// TIA Portal V20 export
// export: Created 2025-12-01T14:57:11.7661616Z, ExportSetting None, DisplayName Totally Integrated Automation Portal, DisplayVersion V20 Update 3, DisplayName TIA Portal Openness, DisplayVersion V20 Update 3, DisplayName TIA Portal Version Control Interface, DisplayVersion V20 Update 3, DisplayName STEP 7 Professional, DisplayVersion V20 Update 3, DisplayName STEP 7 Safety, DisplayVersion V20 Update 2, DisplayName WinCC Basic/Comfort/Advanced, DisplayVersion V20 Update 3, DisplayName WinCC Professional, DisplayVersion V20 Update 3, DisplayName WinCC Unified, DisplayVersion V20 Update 3
FUNCTION "FC920_Registro_Flujos" : Void   // FC920, LAD
TITLE = FC920_Registro_Flujos
{ S7_Optimized_Access := 'FALSE' }
// FC920 Registro Flujos
// stored: AutoNumber false, SetENOAutomatically false
   VAR_INPUT
      Numero_mesa : Int;
   END_VAR
   VAR_TEMP
      cambia_registro : Bool;
      cero : Int;
      retval : Int;
      ROD_CAD : DInt;
      Registro_vacio : Struct
         registro : Array[1..10] of "Registro";
      END_STRUCT;
   END_VAR
   VAR_TEMP   // added for the SCL form of the ladder/FBD networks
      _w1 : Bool;
      _w2 : Bool;
      _w3 : Bool;
      _w4 : Bool;
   END_VAR
BEGIN

REGION Network 1: Inicializacion y cambio de registro registro para poder hacer varios registros
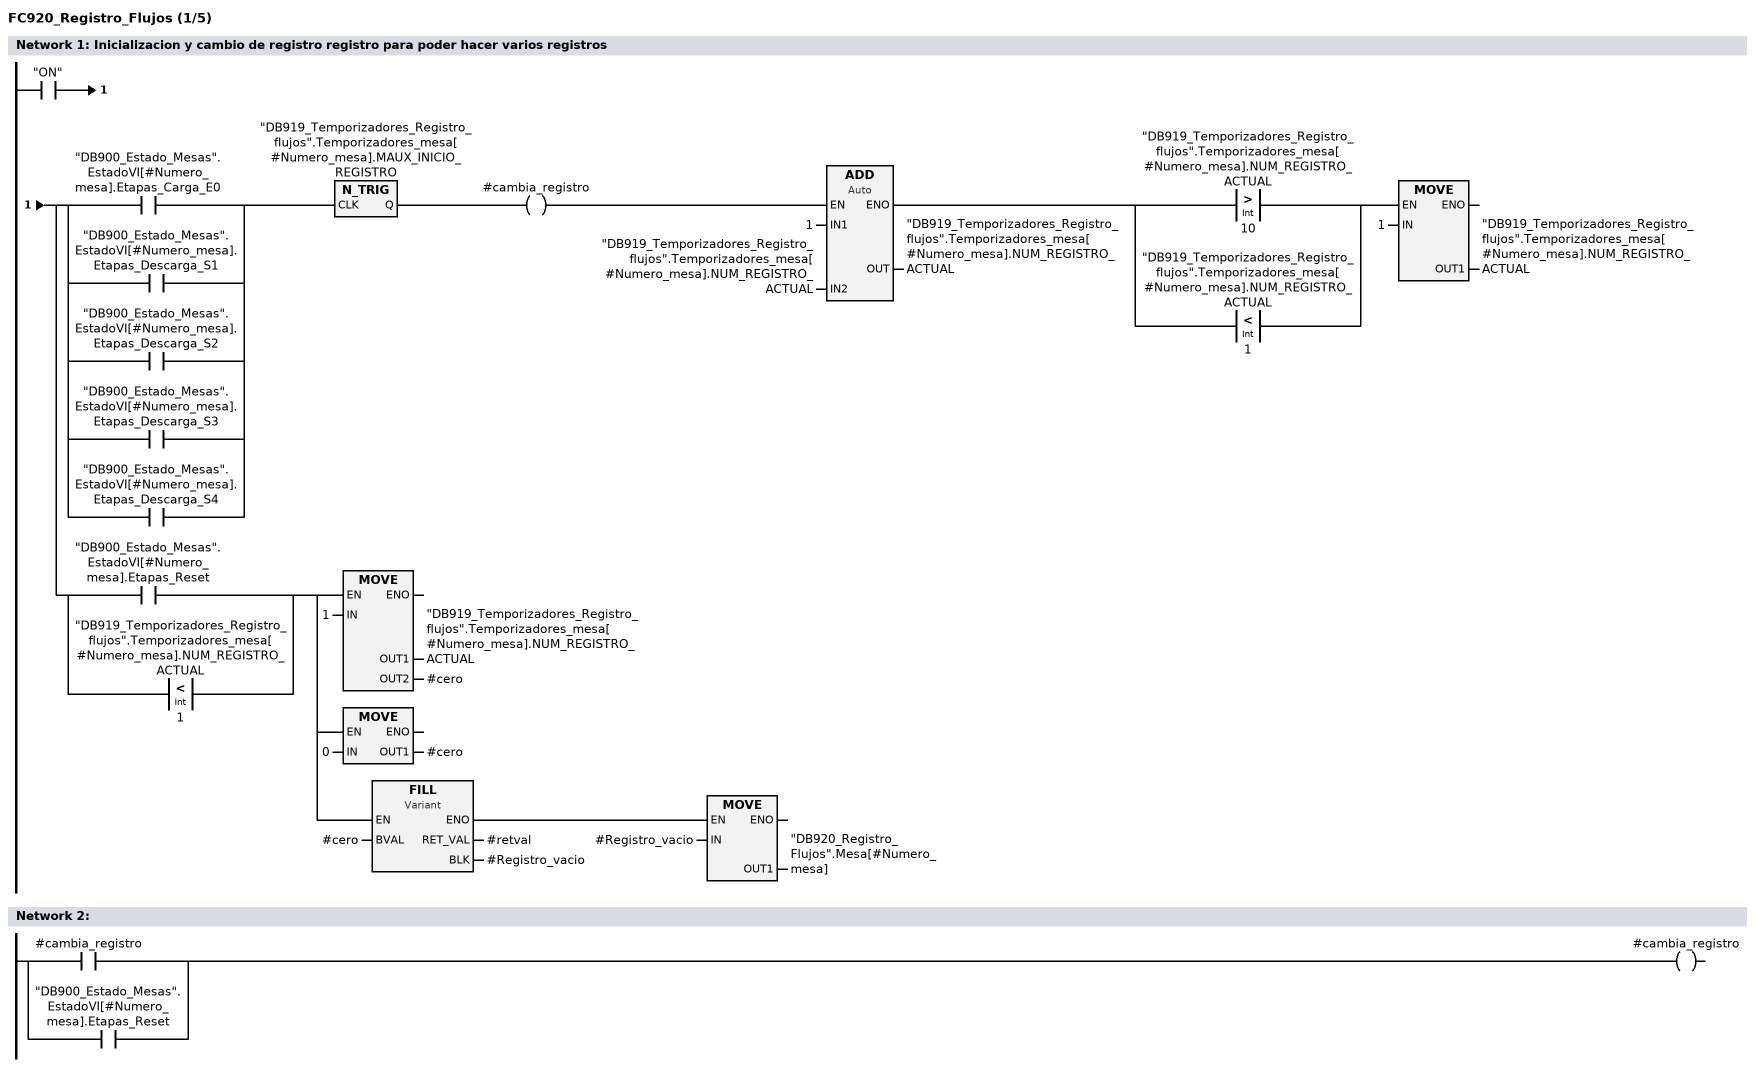
   RUNG wire#powerrail
      Contact( "ON" )
      wire#w1
      Contact( "DB900_Estado_Mesas".EstadoVI[#Numero_mesa].Etapas_Carga_E0 )
      wire#w2
      N_Trig( "DB919_Temporizadores_Registro_flujos".Temporizadores_mesa[#Numero_mesa].MAUX_INICIO_REGISTRO )
      Coil( #cambia_registro )
      Add(in1 := 1, in2 := "DB919_Temporizadores_Registro_flujos".Temporizadores_mesa[#Numero_mesa].NUM_REGISTRO_ACTUAL, out => "DB919_Temporizadores_Registro_flujos".Temporizadores_mesa[#Numero_mesa].NUM_REGISTRO_ACTUAL)
      wire#w3
      { S7_Templates := "SrcType := Int" } GT_Contact(in1 := "DB919_Temporizadores_Registro_flujos".Temporizadores_mesa[#Numero_mesa].NUM_REGISTRO_ACTUAL, in2 := 10)
      wire#w4
      Move(in := 1, out1 => "DB919_Temporizadores_Registro_flujos".Temporizadores_mesa[#Numero_mesa].NUM_REGISTRO_ACTUAL)
   END_RUNG
   RUNG wire#w1
      Contact( "DB900_Estado_Mesas".EstadoVI[#Numero_mesa].Etapas_Descarga_S1 )
   END_RUNG wire#w2
   RUNG wire#w1
      Contact( "DB900_Estado_Mesas".EstadoVI[#Numero_mesa].Etapas_Descarga_S2 )
   END_RUNG wire#w2
   RUNG wire#w1
      Contact( "DB900_Estado_Mesas".EstadoVI[#Numero_mesa].Etapas_Descarga_S3 )
   END_RUNG wire#w2
   RUNG wire#w1
      Contact( "DB900_Estado_Mesas".EstadoVI[#Numero_mesa].Etapas_Descarga_S4 )
   END_RUNG wire#w2
   RUNG wire#w3
      { S7_Templates := "SrcType := Int" } LT_Contact(in1 := "DB919_Temporizadores_Registro_flujos".Temporizadores_mesa[#Numero_mesa].NUM_REGISTRO_ACTUAL, in2 := 1)
   END_RUNG wire#w4
   RUNG wire#w1
      Contact( "DB900_Estado_Mesas".EstadoVI[#Numero_mesa].Etapas_Reset )
      wire#w5
      Move(in := 1, out1 => "DB919_Temporizadores_Registro_flujos".Temporizadores_mesa[#Numero_mesa].NUM_REGISTRO_ACTUAL, out2 => #cero)
   END_RUNG
   RUNG wire#w1
      { S7_Templates := "SrcType := Int" } LT_Contact(in1 := "DB919_Temporizadores_Registro_flujos".Temporizadores_mesa[#Numero_mesa].NUM_REGISTRO_ACTUAL, in2 := 1)
   END_RUNG wire#w5
   RUNG wire#w5
      Move(in := 0, out1 => #cero)
   END_RUNG
   RUNG wire#w5
      { S7_Templates := "ptr_type := Variant" } FILL(BVAL := #cero, RET_VAL => #retval, BLK => #Registro_vacio)
      Move(in := #Registro_vacio, out1 => "DB920_Registro_Flujos".Mesa[#Numero_mesa])
   END_RUNG
   // the same network as SCL:
   #_w1 := "ON" AND ("DB900_Estado_Mesas".EstadoVI[#Numero_mesa].Etapas_Carga_E0 OR "DB900_Estado_Mesas".EstadoVI[#Numero_mesa].Etapas_Descarga_S1 OR "DB900_Estado_Mesas".EstadoVI[#Numero_mesa].Etapas_Descarga_S2 OR "DB900_Estado_Mesas".EstadoVI[#Numero_mesa].Etapas_Descarga_S3 OR "DB900_Estado_Mesas".EstadoVI[#Numero_mesa].Etapas_Descarga_S4);
   #_w2 := NOT #_w1 AND "DB919_Temporizadores_Registro_flujos".Temporizadores_mesa[#Numero_mesa].MAUX_INICIO_REGISTRO;   // falling edge
   "DB919_Temporizadores_Registro_flujos".Temporizadores_mesa[#Numero_mesa].MAUX_INICIO_REGISTRO := #_w1;
   #cambia_registro := #_w2;
   IF #_w2 THEN
       "DB919_Temporizadores_Registro_flujos".Temporizadores_mesa[#Numero_mesa].NUM_REGISTRO_ACTUAL := 1 + "DB919_Temporizadores_Registro_flujos".Temporizadores_mesa[#Numero_mesa].NUM_REGISTRO_ACTUAL;
   END_IF;
   IF #_w2 AND (("DB919_Temporizadores_Registro_flujos".Temporizadores_mesa[#Numero_mesa].NUM_REGISTRO_ACTUAL > 10) OR ("DB919_Temporizadores_Registro_flujos".Temporizadores_mesa[#Numero_mesa].NUM_REGISTRO_ACTUAL < 1)) THEN
       "DB919_Temporizadores_Registro_flujos".Temporizadores_mesa[#Numero_mesa].NUM_REGISTRO_ACTUAL := 1;
   END_IF;
   #_w3 := "ON" AND ("DB900_Estado_Mesas".EstadoVI[#Numero_mesa].Etapas_Reset OR ("DB919_Temporizadores_Registro_flujos".Temporizadores_mesa[#Numero_mesa].NUM_REGISTRO_ACTUAL < 1));
   IF #_w3 THEN
       "DB919_Temporizadores_Registro_flujos".Temporizadores_mesa[#Numero_mesa].NUM_REGISTRO_ACTUAL := 1;
       #cero := 1;
       #cero := 0;
   END_IF;
   #retval := FILL(EN := #_w3, BVAL := #cero, BLK => #Registro_vacio, ENO => #_w4);
   IF #_w4 THEN "DB920_Registro_Flujos".Mesa[#Numero_mesa] := #Registro_vacio; END_IF;
END_REGION

REGION Network 2
   RUNG wire#powerrail
      Contact( #cambia_registro )
      wire#w1
      Coil( #cambia_registro )
   END_RUNG
   RUNG wire#powerrail
      Contact( "DB900_Estado_Mesas".EstadoVI[#Numero_mesa].Etapas_Reset )
   END_RUNG wire#w1
   // the same network as SCL:
   #cambia_registro := #cambia_registro OR "DB900_Estado_Mesas".EstadoVI[#Numero_mesa].Etapas_Reset;
END_REGION

REGION Network 3: Temporizador Etapas de Carga
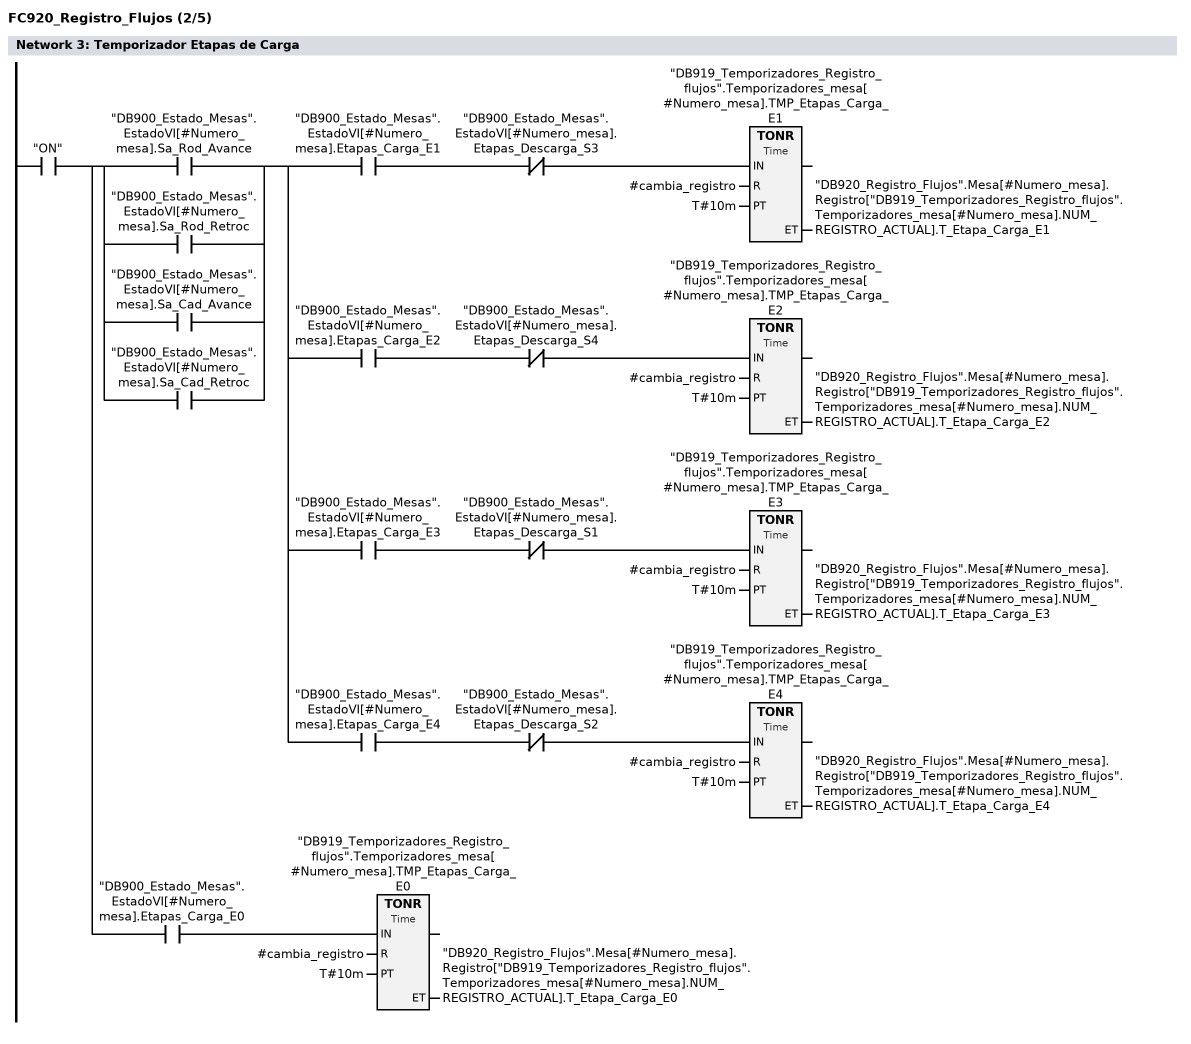
   RUNG wire#powerrail
      Contact( "ON" )
      wire#w1
      Contact( "DB900_Estado_Mesas".EstadoVI[#Numero_mesa].Sa_Rod_Avance )
      wire#w2
      Contact( "DB900_Estado_Mesas".EstadoVI[#Numero_mesa].Etapas_Carga_E1 )
      I_Contact( "DB900_Estado_Mesas".EstadoVI[#Numero_mesa].Etapas_Descarga_S3 )
      { S7_Templates := "time_type := Time" } "DB919_Temporizadores_Registro_flujos".Temporizadores_mesa[#Numero_mesa].TMP_Etapas_Carga_E1.TONR(r := #cambia_registro, pt := T#10m, et => "DB920_Registro_Flujos".Mesa[#Numero_mesa].Registro["DB919_Temporizadores_Registro_flujos".Temporizadores_mesa[#Numero_mesa].NUM_REGISTRO_ACTUAL].T_Etapa_Carga_E1)
   END_RUNG
   RUNG wire#w1
      Contact( "DB900_Estado_Mesas".EstadoVI[#Numero_mesa].Sa_Rod_Retroc )
   END_RUNG wire#w2
   RUNG wire#w1
      Contact( "DB900_Estado_Mesas".EstadoVI[#Numero_mesa].Sa_Cad_Avance )
   END_RUNG wire#w2
   RUNG wire#w1
      Contact( "DB900_Estado_Mesas".EstadoVI[#Numero_mesa].Sa_Cad_Retroc )
   END_RUNG wire#w2
   RUNG wire#w2
      Contact( "DB900_Estado_Mesas".EstadoVI[#Numero_mesa].Etapas_Carga_E2 )
      I_Contact( "DB900_Estado_Mesas".EstadoVI[#Numero_mesa].Etapas_Descarga_S4 )
      { S7_Templates := "time_type := Time" } "DB919_Temporizadores_Registro_flujos".Temporizadores_mesa[#Numero_mesa].TMP_Etapas_Carga_E2.TONR(r := #cambia_registro, pt := T#10m, et => "DB920_Registro_Flujos".Mesa[#Numero_mesa].Registro["DB919_Temporizadores_Registro_flujos".Temporizadores_mesa[#Numero_mesa].NUM_REGISTRO_ACTUAL].T_Etapa_Carga_E2)
   END_RUNG
   RUNG wire#w2
      Contact( "DB900_Estado_Mesas".EstadoVI[#Numero_mesa].Etapas_Carga_E3 )
      I_Contact( "DB900_Estado_Mesas".EstadoVI[#Numero_mesa].Etapas_Descarga_S1 )
      { S7_Templates := "time_type := Time" } "DB919_Temporizadores_Registro_flujos".Temporizadores_mesa[#Numero_mesa].TMP_Etapas_Carga_E3.TONR(r := #cambia_registro, pt := T#10m, et => "DB920_Registro_Flujos".Mesa[#Numero_mesa].Registro["DB919_Temporizadores_Registro_flujos".Temporizadores_mesa[#Numero_mesa].NUM_REGISTRO_ACTUAL].T_Etapa_Carga_E3)
   END_RUNG
   RUNG wire#w2
      Contact( "DB900_Estado_Mesas".EstadoVI[#Numero_mesa].Etapas_Carga_E4 )
      I_Contact( "DB900_Estado_Mesas".EstadoVI[#Numero_mesa].Etapas_Descarga_S2 )
      { S7_Templates := "time_type := Time" } "DB919_Temporizadores_Registro_flujos".Temporizadores_mesa[#Numero_mesa].TMP_Etapas_Carga_E4.TONR(r := #cambia_registro, pt := T#10m, et => "DB920_Registro_Flujos".Mesa[#Numero_mesa].Registro["DB919_Temporizadores_Registro_flujos".Temporizadores_mesa[#Numero_mesa].NUM_REGISTRO_ACTUAL].T_Etapa_Carga_E4)
   END_RUNG
   RUNG wire#w1
      Contact( "DB900_Estado_Mesas".EstadoVI[#Numero_mesa].Etapas_Carga_E0 )
      { S7_Templates := "time_type := Time" } "DB919_Temporizadores_Registro_flujos".Temporizadores_mesa[#Numero_mesa].TMP_Etapas_Carga_E0.TONR(r := #cambia_registro, pt := T#10m, et => "DB920_Registro_Flujos".Mesa[#Numero_mesa].Registro["DB919_Temporizadores_Registro_flujos".Temporizadores_mesa[#Numero_mesa].NUM_REGISTRO_ACTUAL].T_Etapa_Carga_E0)
   END_RUNG
   // the same network as SCL:
   #_w1 := "ON" AND ("DB900_Estado_Mesas".EstadoVI[#Numero_mesa].Sa_Rod_Avance OR "DB900_Estado_Mesas".EstadoVI[#Numero_mesa].Sa_Rod_Retroc OR "DB900_Estado_Mesas".EstadoVI[#Numero_mesa].Sa_Cad_Avance OR "DB900_Estado_Mesas".EstadoVI[#Numero_mesa].Sa_Cad_Retroc);
   "DB919_Temporizadores_Registro_flujos".Temporizadores_mesa[#Numero_mesa].TMP_Etapas_Carga_E1.TONR(IN := #_w1 AND "DB900_Estado_Mesas".EstadoVI[#Numero_mesa].Etapas_Carga_E1 AND NOT "DB900_Estado_Mesas".EstadoVI[#Numero_mesa].Etapas_Descarga_S3,
                           R := #cambia_registro,
                           PT := T#10m,
                           ET => "DB920_Registro_Flujos".Mesa[#Numero_mesa].Registro["DB919_Temporizadores_Registro_flujos".Temporizadores_mesa[#Numero_mesa].NUM_REGISTRO_ACTUAL].T_Etapa_Carga_E1);
   "DB919_Temporizadores_Registro_flujos".Temporizadores_mesa[#Numero_mesa].TMP_Etapas_Carga_E2.TONR(IN := #_w1 AND "DB900_Estado_Mesas".EstadoVI[#Numero_mesa].Etapas_Carga_E2 AND NOT "DB900_Estado_Mesas".EstadoVI[#Numero_mesa].Etapas_Descarga_S4,
                           R := #cambia_registro,
                           PT := T#10m,
                           ET => "DB920_Registro_Flujos".Mesa[#Numero_mesa].Registro["DB919_Temporizadores_Registro_flujos".Temporizadores_mesa[#Numero_mesa].NUM_REGISTRO_ACTUAL].T_Etapa_Carga_E2);
   "DB919_Temporizadores_Registro_flujos".Temporizadores_mesa[#Numero_mesa].TMP_Etapas_Carga_E3.TONR(IN := #_w1 AND "DB900_Estado_Mesas".EstadoVI[#Numero_mesa].Etapas_Carga_E3 AND NOT "DB900_Estado_Mesas".EstadoVI[#Numero_mesa].Etapas_Descarga_S1,
                           R := #cambia_registro,
                           PT := T#10m,
                           ET => "DB920_Registro_Flujos".Mesa[#Numero_mesa].Registro["DB919_Temporizadores_Registro_flujos".Temporizadores_mesa[#Numero_mesa].NUM_REGISTRO_ACTUAL].T_Etapa_Carga_E3);
   "DB919_Temporizadores_Registro_flujos".Temporizadores_mesa[#Numero_mesa].TMP_Etapas_Carga_E4.TONR(IN := #_w1 AND "DB900_Estado_Mesas".EstadoVI[#Numero_mesa].Etapas_Carga_E4 AND NOT "DB900_Estado_Mesas".EstadoVI[#Numero_mesa].Etapas_Descarga_S2,
                           R := #cambia_registro,
                           PT := T#10m,
                           ET => "DB920_Registro_Flujos".Mesa[#Numero_mesa].Registro["DB919_Temporizadores_Registro_flujos".Temporizadores_mesa[#Numero_mesa].NUM_REGISTRO_ACTUAL].T_Etapa_Carga_E4);
   "DB919_Temporizadores_Registro_flujos".Temporizadores_mesa[#Numero_mesa].TMP_Etapas_Carga_E0.TONR(IN := "ON" AND "DB900_Estado_Mesas".EstadoVI[#Numero_mesa].Etapas_Carga_E0,
                           R := #cambia_registro,
                           PT := T#10m,
                           ET => "DB920_Registro_Flujos".Mesa[#Numero_mesa].Registro["DB919_Temporizadores_Registro_flujos".Temporizadores_mesa[#Numero_mesa].NUM_REGISTRO_ACTUAL].T_Etapa_Carga_E0);
END_REGION

REGION Network 4: Temporizador Etapas de Descarga
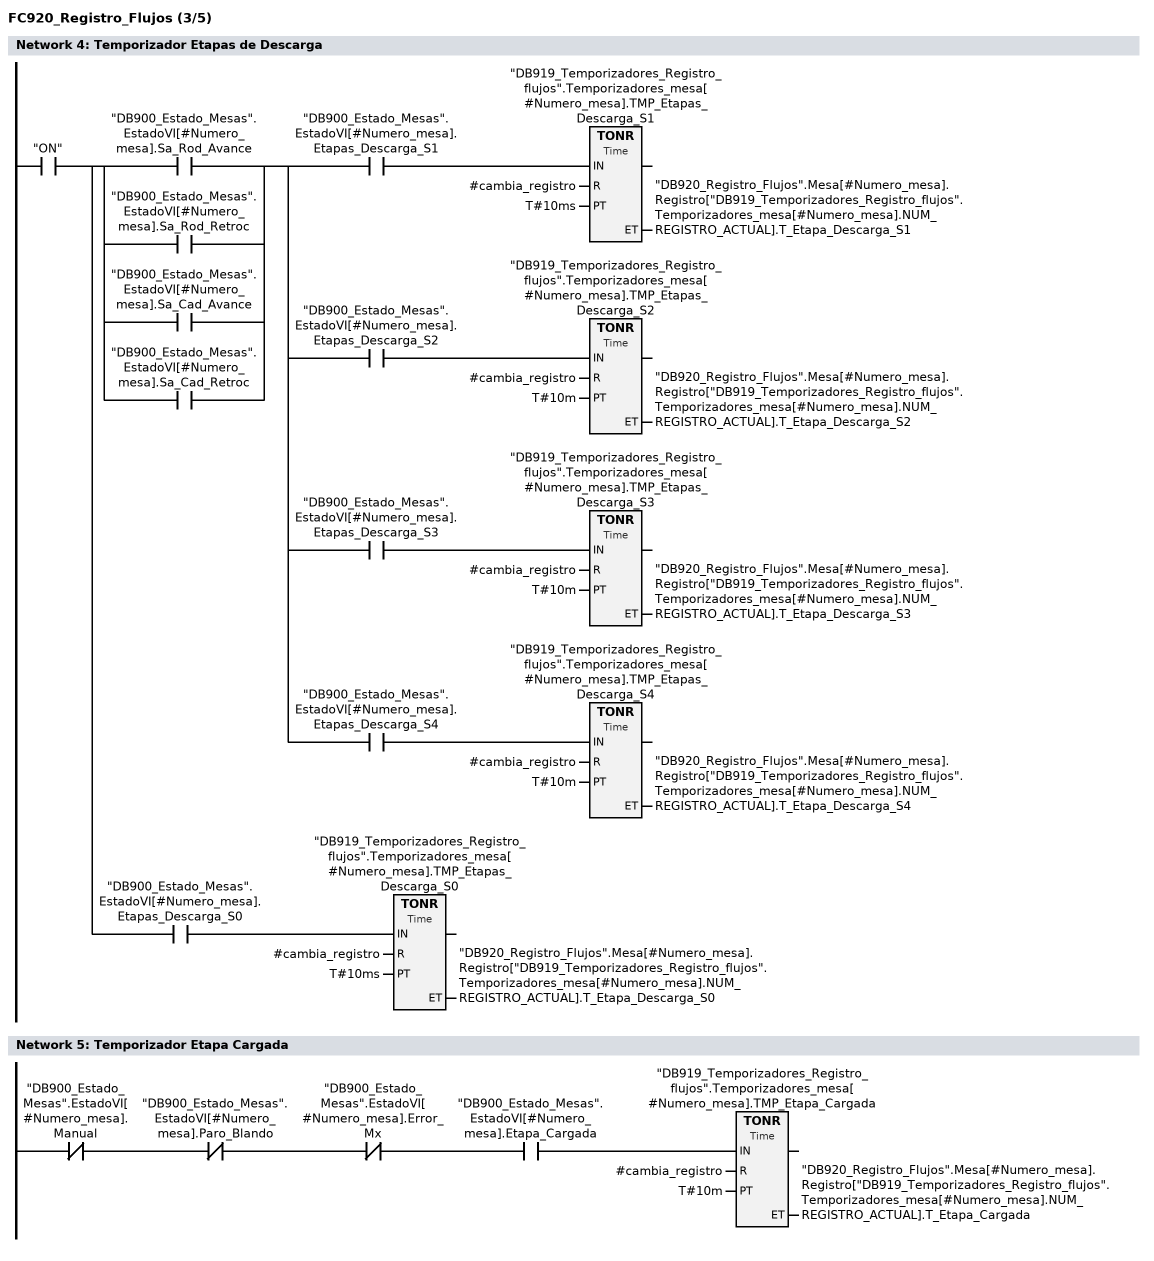
   RUNG wire#powerrail
      Contact( "ON" )
      wire#w1
      Contact( "DB900_Estado_Mesas".EstadoVI[#Numero_mesa].Sa_Rod_Avance )
      wire#w2
      Contact( "DB900_Estado_Mesas".EstadoVI[#Numero_mesa].Etapas_Descarga_S1 )
      { S7_Templates := "time_type := Time" } "DB919_Temporizadores_Registro_flujos".Temporizadores_mesa[#Numero_mesa].TMP_Etapas_Descarga_S1.TONR(r := #cambia_registro, pt := T#10ms, et => "DB920_Registro_Flujos".Mesa[#Numero_mesa].Registro["DB919_Temporizadores_Registro_flujos".Temporizadores_mesa[#Numero_mesa].NUM_REGISTRO_ACTUAL].T_Etapa_Descarga_S1)
   END_RUNG
   RUNG wire#w1
      Contact( "DB900_Estado_Mesas".EstadoVI[#Numero_mesa].Sa_Rod_Retroc )
   END_RUNG wire#w2
   RUNG wire#w1
      Contact( "DB900_Estado_Mesas".EstadoVI[#Numero_mesa].Sa_Cad_Avance )
   END_RUNG wire#w2
   RUNG wire#w1
      Contact( "DB900_Estado_Mesas".EstadoVI[#Numero_mesa].Sa_Cad_Retroc )
   END_RUNG wire#w2
   RUNG wire#w2
      Contact( "DB900_Estado_Mesas".EstadoVI[#Numero_mesa].Etapas_Descarga_S2 )
      { S7_Templates := "time_type := Time" } "DB919_Temporizadores_Registro_flujos".Temporizadores_mesa[#Numero_mesa].TMP_Etapas_Descarga_S2.TONR(r := #cambia_registro, pt := T#10m, et => "DB920_Registro_Flujos".Mesa[#Numero_mesa].Registro["DB919_Temporizadores_Registro_flujos".Temporizadores_mesa[#Numero_mesa].NUM_REGISTRO_ACTUAL].T_Etapa_Descarga_S2)
   END_RUNG
   RUNG wire#w2
      Contact( "DB900_Estado_Mesas".EstadoVI[#Numero_mesa].Etapas_Descarga_S3 )
      { S7_Templates := "time_type := Time" } "DB919_Temporizadores_Registro_flujos".Temporizadores_mesa[#Numero_mesa].TMP_Etapas_Descarga_S3.TONR(r := #cambia_registro, pt := T#10m, et => "DB920_Registro_Flujos".Mesa[#Numero_mesa].Registro["DB919_Temporizadores_Registro_flujos".Temporizadores_mesa[#Numero_mesa].NUM_REGISTRO_ACTUAL].T_Etapa_Descarga_S3)
   END_RUNG
   RUNG wire#w2
      Contact( "DB900_Estado_Mesas".EstadoVI[#Numero_mesa].Etapas_Descarga_S4 )
      { S7_Templates := "time_type := Time" } "DB919_Temporizadores_Registro_flujos".Temporizadores_mesa[#Numero_mesa].TMP_Etapas_Descarga_S4.TONR(r := #cambia_registro, pt := T#10m, et => "DB920_Registro_Flujos".Mesa[#Numero_mesa].Registro["DB919_Temporizadores_Registro_flujos".Temporizadores_mesa[#Numero_mesa].NUM_REGISTRO_ACTUAL].T_Etapa_Descarga_S4)
   END_RUNG
   RUNG wire#w1
      Contact( "DB900_Estado_Mesas".EstadoVI[#Numero_mesa].Etapas_Descarga_S0 )
      { S7_Templates := "time_type := Time" } "DB919_Temporizadores_Registro_flujos".Temporizadores_mesa[#Numero_mesa].TMP_Etapas_Descarga_S0.TONR(r := #cambia_registro, pt := T#10ms, et => "DB920_Registro_Flujos".Mesa[#Numero_mesa].Registro["DB919_Temporizadores_Registro_flujos".Temporizadores_mesa[#Numero_mesa].NUM_REGISTRO_ACTUAL].T_Etapa_Descarga_S0)
   END_RUNG
   // the same network as SCL:
   #_w1 := "ON" AND ("DB900_Estado_Mesas".EstadoVI[#Numero_mesa].Sa_Rod_Avance OR "DB900_Estado_Mesas".EstadoVI[#Numero_mesa].Sa_Rod_Retroc OR "DB900_Estado_Mesas".EstadoVI[#Numero_mesa].Sa_Cad_Avance OR "DB900_Estado_Mesas".EstadoVI[#Numero_mesa].Sa_Cad_Retroc);
   "DB919_Temporizadores_Registro_flujos".Temporizadores_mesa[#Numero_mesa].TMP_Etapas_Descarga_S1.TONR(IN := #_w1 AND "DB900_Estado_Mesas".EstadoVI[#Numero_mesa].Etapas_Descarga_S1,
                           R := #cambia_registro,
                           PT := T#10ms,
                           ET => "DB920_Registro_Flujos".Mesa[#Numero_mesa].Registro["DB919_Temporizadores_Registro_flujos".Temporizadores_mesa[#Numero_mesa].NUM_REGISTRO_ACTUAL].T_Etapa_Descarga_S1);
   "DB919_Temporizadores_Registro_flujos".Temporizadores_mesa[#Numero_mesa].TMP_Etapas_Descarga_S2.TONR(IN := #_w1 AND "DB900_Estado_Mesas".EstadoVI[#Numero_mesa].Etapas_Descarga_S2,
                           R := #cambia_registro,
                           PT := T#10m,
                           ET => "DB920_Registro_Flujos".Mesa[#Numero_mesa].Registro["DB919_Temporizadores_Registro_flujos".Temporizadores_mesa[#Numero_mesa].NUM_REGISTRO_ACTUAL].T_Etapa_Descarga_S2);
   "DB919_Temporizadores_Registro_flujos".Temporizadores_mesa[#Numero_mesa].TMP_Etapas_Descarga_S3.TONR(IN := #_w1 AND "DB900_Estado_Mesas".EstadoVI[#Numero_mesa].Etapas_Descarga_S3,
                           R := #cambia_registro,
                           PT := T#10m,
                           ET => "DB920_Registro_Flujos".Mesa[#Numero_mesa].Registro["DB919_Temporizadores_Registro_flujos".Temporizadores_mesa[#Numero_mesa].NUM_REGISTRO_ACTUAL].T_Etapa_Descarga_S3);
   "DB919_Temporizadores_Registro_flujos".Temporizadores_mesa[#Numero_mesa].TMP_Etapas_Descarga_S4.TONR(IN := #_w1 AND "DB900_Estado_Mesas".EstadoVI[#Numero_mesa].Etapas_Descarga_S4,
                           R := #cambia_registro,
                           PT := T#10m,
                           ET => "DB920_Registro_Flujos".Mesa[#Numero_mesa].Registro["DB919_Temporizadores_Registro_flujos".Temporizadores_mesa[#Numero_mesa].NUM_REGISTRO_ACTUAL].T_Etapa_Descarga_S4);
   "DB919_Temporizadores_Registro_flujos".Temporizadores_mesa[#Numero_mesa].TMP_Etapas_Descarga_S0.TONR(IN := "ON" AND "DB900_Estado_Mesas".EstadoVI[#Numero_mesa].Etapas_Descarga_S0,
                           R := #cambia_registro,
                           PT := T#10ms,
                           ET => "DB920_Registro_Flujos".Mesa[#Numero_mesa].Registro["DB919_Temporizadores_Registro_flujos".Temporizadores_mesa[#Numero_mesa].NUM_REGISTRO_ACTUAL].T_Etapa_Descarga_S0);
END_REGION

REGION Network 5: Temporizador Etapa Cargada
   RUNG wire#powerrail
      I_Contact( "DB900_Estado_Mesas".EstadoVI[#Numero_mesa].Manual )
      I_Contact( "DB900_Estado_Mesas".EstadoVI[#Numero_mesa].Paro_Blando )
      I_Contact( "DB900_Estado_Mesas".EstadoVI[#Numero_mesa].Error_Mx )
      Contact( "DB900_Estado_Mesas".EstadoVI[#Numero_mesa].Etapa_Cargada )
      { S7_Templates := "time_type := Time" } "DB919_Temporizadores_Registro_flujos".Temporizadores_mesa[#Numero_mesa].TMP_Etapa_Cargada.TONR(r := #cambia_registro, pt := T#10m, et => "DB920_Registro_Flujos".Mesa[#Numero_mesa].Registro["DB919_Temporizadores_Registro_flujos".Temporizadores_mesa[#Numero_mesa].NUM_REGISTRO_ACTUAL].T_Etapa_Cargada)
   END_RUNG
   // the same network as SCL:
   "DB919_Temporizadores_Registro_flujos".Temporizadores_mesa[#Numero_mesa].TMP_Etapa_Cargada.TONR(IN := NOT "DB900_Estado_Mesas".EstadoVI[#Numero_mesa].Manual AND NOT "DB900_Estado_Mesas".EstadoVI[#Numero_mesa].Paro_Blando AND NOT "DB900_Estado_Mesas".EstadoVI[#Numero_mesa].Error_Mx AND "DB900_Estado_Mesas".EstadoVI[#Numero_mesa].Etapa_Cargada,
                           R := #cambia_registro,
                           PT := T#10m,
                           ET => "DB920_Registro_Flujos".Mesa[#Numero_mesa].Registro["DB919_Temporizadores_Registro_flujos".Temporizadores_mesa[#Numero_mesa].NUM_REGISTRO_ACTUAL].T_Etapa_Cargada);
END_REGION

REGION Network 6: Temporizador Avance/Retroceso Rodillos
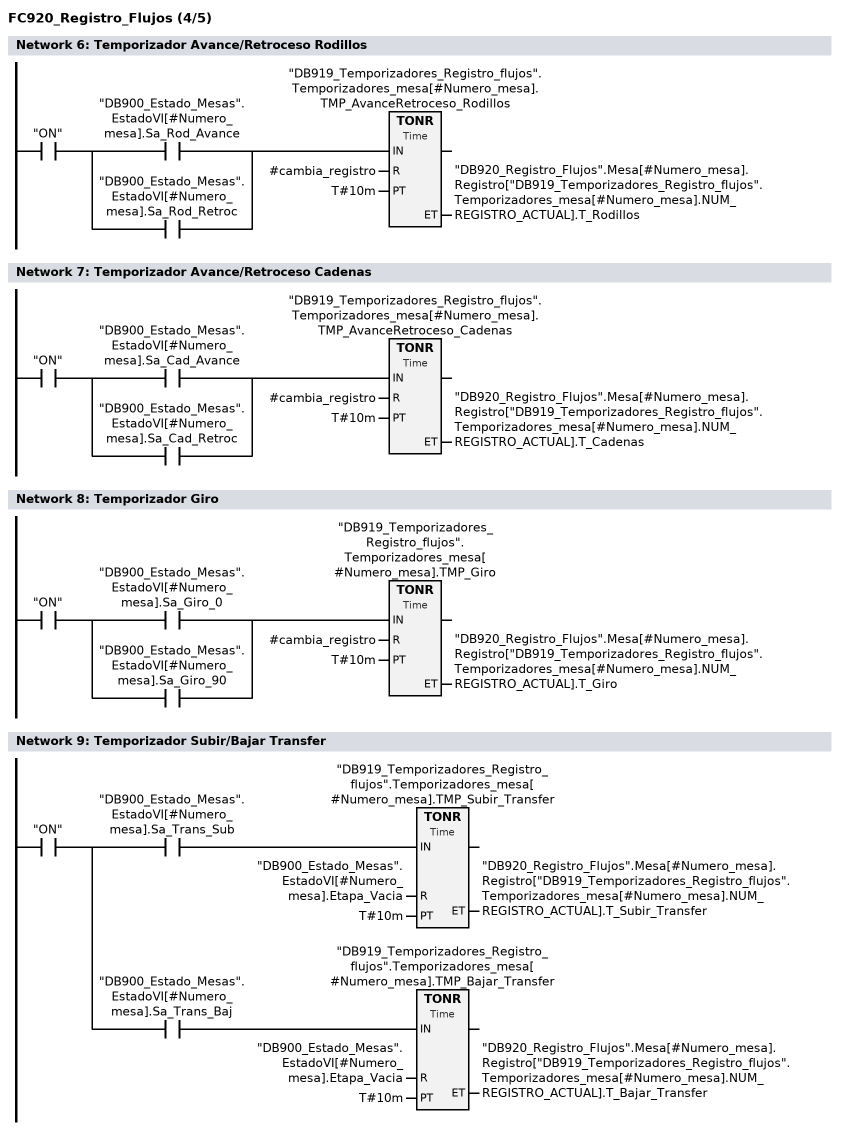
   RUNG wire#powerrail
      Contact( "ON" )
      wire#w1
      Contact( "DB900_Estado_Mesas".EstadoVI[#Numero_mesa].Sa_Rod_Avance )
      wire#w2
      { S7_Templates := "time_type := Time" } "DB919_Temporizadores_Registro_flujos".Temporizadores_mesa[#Numero_mesa].TMP_AvanceRetroceso_Rodillos.TONR(r := #cambia_registro, pt := T#10m, et => "DB920_Registro_Flujos".Mesa[#Numero_mesa].Registro["DB919_Temporizadores_Registro_flujos".Temporizadores_mesa[#Numero_mesa].NUM_REGISTRO_ACTUAL].T_Rodillos)
   END_RUNG
   RUNG wire#w1
      Contact( "DB900_Estado_Mesas".EstadoVI[#Numero_mesa].Sa_Rod_Retroc )
   END_RUNG wire#w2
   // the same network as SCL:
   "DB919_Temporizadores_Registro_flujos".Temporizadores_mesa[#Numero_mesa].TMP_AvanceRetroceso_Rodillos.TONR(IN := "ON" AND ("DB900_Estado_Mesas".EstadoVI[#Numero_mesa].Sa_Rod_Avance OR "DB900_Estado_Mesas".EstadoVI[#Numero_mesa].Sa_Rod_Retroc),
                           R := #cambia_registro,
                           PT := T#10m,
                           ET => "DB920_Registro_Flujos".Mesa[#Numero_mesa].Registro["DB919_Temporizadores_Registro_flujos".Temporizadores_mesa[#Numero_mesa].NUM_REGISTRO_ACTUAL].T_Rodillos);
END_REGION

REGION Network 7: Temporizador Avance/Retroceso Cadenas
   RUNG wire#powerrail
      Contact( "ON" )
      wire#w1
      Contact( "DB900_Estado_Mesas".EstadoVI[#Numero_mesa].Sa_Cad_Avance )
      wire#w2
      { S7_Templates := "time_type := Time" } "DB919_Temporizadores_Registro_flujos".Temporizadores_mesa[#Numero_mesa].TMP_AvanceRetroceso_Cadenas.TONR(r := #cambia_registro, pt := T#10m, et => "DB920_Registro_Flujos".Mesa[#Numero_mesa].Registro["DB919_Temporizadores_Registro_flujos".Temporizadores_mesa[#Numero_mesa].NUM_REGISTRO_ACTUAL].T_Cadenas)
   END_RUNG
   RUNG wire#w1
      Contact( "DB900_Estado_Mesas".EstadoVI[#Numero_mesa].Sa_Cad_Retroc )
   END_RUNG wire#w2
   // the same network as SCL:
   "DB919_Temporizadores_Registro_flujos".Temporizadores_mesa[#Numero_mesa].TMP_AvanceRetroceso_Cadenas.TONR(IN := "ON" AND ("DB900_Estado_Mesas".EstadoVI[#Numero_mesa].Sa_Cad_Avance OR "DB900_Estado_Mesas".EstadoVI[#Numero_mesa].Sa_Cad_Retroc),
                           R := #cambia_registro,
                           PT := T#10m,
                           ET => "DB920_Registro_Flujos".Mesa[#Numero_mesa].Registro["DB919_Temporizadores_Registro_flujos".Temporizadores_mesa[#Numero_mesa].NUM_REGISTRO_ACTUAL].T_Cadenas);
END_REGION

REGION Network 8: Temporizador Giro
   RUNG wire#powerrail
      Contact( "ON" )
      wire#w1
      Contact( "DB900_Estado_Mesas".EstadoVI[#Numero_mesa].Sa_Giro_0 )
      wire#w2
      { S7_Templates := "time_type := Time" } "DB919_Temporizadores_Registro_flujos".Temporizadores_mesa[#Numero_mesa].TMP_Giro.TONR(r := #cambia_registro, pt := T#10m, et => "DB920_Registro_Flujos".Mesa[#Numero_mesa].Registro["DB919_Temporizadores_Registro_flujos".Temporizadores_mesa[#Numero_mesa].NUM_REGISTRO_ACTUAL].T_Giro)
   END_RUNG
   RUNG wire#w1
      Contact( "DB900_Estado_Mesas".EstadoVI[#Numero_mesa].Sa_Giro_90 )
   END_RUNG wire#w2
   // the same network as SCL:
   "DB919_Temporizadores_Registro_flujos".Temporizadores_mesa[#Numero_mesa].TMP_Giro.TONR(IN := "ON" AND ("DB900_Estado_Mesas".EstadoVI[#Numero_mesa].Sa_Giro_0 OR "DB900_Estado_Mesas".EstadoVI[#Numero_mesa].Sa_Giro_90),
                           R := #cambia_registro,
                           PT := T#10m,
                           ET => "DB920_Registro_Flujos".Mesa[#Numero_mesa].Registro["DB919_Temporizadores_Registro_flujos".Temporizadores_mesa[#Numero_mesa].NUM_REGISTRO_ACTUAL].T_Giro);
END_REGION

REGION Network 9: Temporizador Subir/Bajar Transfer
   RUNG wire#powerrail
      Contact( "ON" )
      wire#w1
      Contact( "DB900_Estado_Mesas".EstadoVI[#Numero_mesa].Sa_Trans_Sub )
      { S7_Templates := "time_type := Time" } "DB919_Temporizadores_Registro_flujos".Temporizadores_mesa[#Numero_mesa].TMP_Subir_Transfer.TONR(r := "DB900_Estado_Mesas".EstadoVI[#Numero_mesa].Etapa_Vacia, pt := T#10m, et => "DB920_Registro_Flujos".Mesa[#Numero_mesa].Registro["DB919_Temporizadores_Registro_flujos".Temporizadores_mesa[#Numero_mesa].NUM_REGISTRO_ACTUAL].T_Subir_Transfer)
   END_RUNG
   RUNG wire#w1
      Contact( "DB900_Estado_Mesas".EstadoVI[#Numero_mesa].Sa_Trans_Baj )
      { S7_Templates := "time_type := Time" } "DB919_Temporizadores_Registro_flujos".Temporizadores_mesa[#Numero_mesa].TMP_Bajar_Transfer.TONR(r := "DB900_Estado_Mesas".EstadoVI[#Numero_mesa].Etapa_Vacia, pt := T#10m, et => "DB920_Registro_Flujos".Mesa[#Numero_mesa].Registro["DB919_Temporizadores_Registro_flujos".Temporizadores_mesa[#Numero_mesa].NUM_REGISTRO_ACTUAL].T_Bajar_Transfer)
   END_RUNG
   // the same network as SCL:
   "DB919_Temporizadores_Registro_flujos".Temporizadores_mesa[#Numero_mesa].TMP_Subir_Transfer.TONR(IN := "ON" AND "DB900_Estado_Mesas".EstadoVI[#Numero_mesa].Sa_Trans_Sub,
                           R := "DB900_Estado_Mesas".EstadoVI[#Numero_mesa].Etapa_Vacia,
                           PT := T#10m,
                           ET => "DB920_Registro_Flujos".Mesa[#Numero_mesa].Registro["DB919_Temporizadores_Registro_flujos".Temporizadores_mesa[#Numero_mesa].NUM_REGISTRO_ACTUAL].T_Subir_Transfer);
   "DB919_Temporizadores_Registro_flujos".Temporizadores_mesa[#Numero_mesa].TMP_Bajar_Transfer.TONR(IN := "ON" AND "DB900_Estado_Mesas".EstadoVI[#Numero_mesa].Sa_Trans_Baj,
                           R := "DB900_Estado_Mesas".EstadoVI[#Numero_mesa].Etapa_Vacia,
                           PT := T#10m,
                           ET => "DB920_Registro_Flujos".Mesa[#Numero_mesa].Registro["DB919_Temporizadores_Registro_flujos".Temporizadores_mesa[#Numero_mesa].NUM_REGISTRO_ACTUAL].T_Bajar_Transfer);
END_REGION

REGION Network 10: Temporizador TOTAL
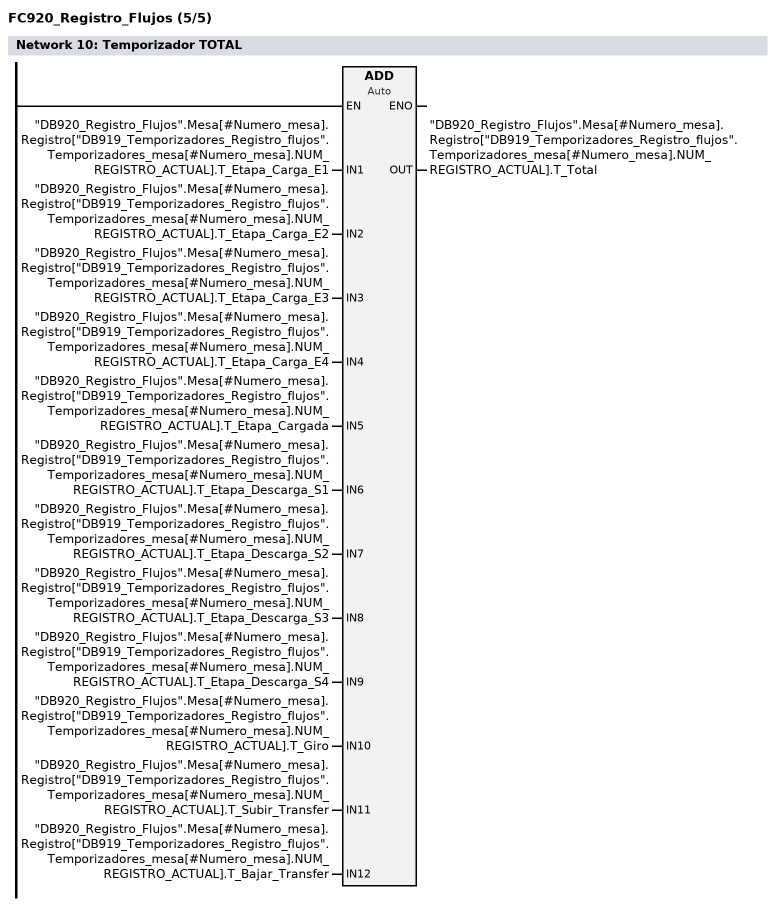
   RUNG wire#powerrail
      Add(in1 := "DB920_Registro_Flujos".Mesa[#Numero_mesa].Registro["DB919_Temporizadores_Registro_flujos".Temporizadores_mesa[#Numero_mesa].NUM_REGISTRO_ACTUAL].T_Etapa_Carga_E1, in2 := "DB920_Registro_Flujos".Mesa[#Numero_mesa].Registro["DB919_Temporizadores_Registro_flujos".Temporizadores_mesa[#Numero_mesa].NUM_REGISTRO_ACTUAL].T_Etapa_Carga_E2, in3 := "DB920_Registro_Flujos".Mesa[#Numero_mesa].Registro["DB919_Temporizadores_Registro_flujos".Temporizadores_mesa[#Numero_mesa].NUM_REGISTRO_ACTUAL].T_Etapa_Carga_E3, in4 := "DB920_Registro_Flujos".Mesa[#Numero_mesa].Registro["DB919_Temporizadores_Registro_flujos".Temporizadores_mesa[#Numero_mesa].NUM_REGISTRO_ACTUAL].T_Etapa_Carga_E4, in5 := "DB920_Registro_Flujos".Mesa[#Numero_mesa].Registro["DB919_Temporizadores_Registro_flujos".Temporizadores_mesa[#Numero_mesa].NUM_REGISTRO_ACTUAL].T_Etapa_Cargada, in6 := "DB920_Registro_Flujos".Mesa[#Numero_mesa].Registro["DB919_Temporizadores_Registro_flujos".Temporizadores_mesa[#Numero_mesa].NUM_REGISTRO_ACTUAL].T_Etapa_Descarga_S1, in7 := "DB920_Registro_Flujos".Mesa[#Numero_mesa].Registro["DB919_Temporizadores_Registro_flujos".Temporizadores_mesa[#Numero_mesa].NUM_REGISTRO_ACTUAL].T_Etapa_Descarga_S2, in8 := "DB920_Registro_Flujos".Mesa[#Numero_mesa].Registro["DB919_Temporizadores_Registro_flujos".Temporizadores_mesa[#Numero_mesa].NUM_REGISTRO_ACTUAL].T_Etapa_Descarga_S3, in9 := "DB920_Registro_Flujos".Mesa[#Numero_mesa].Registro["DB919_Temporizadores_Registro_flujos".Temporizadores_mesa[#Numero_mesa].NUM_REGISTRO_ACTUAL].T_Etapa_Descarga_S4, in10 := "DB920_Registro_Flujos".Mesa[#Numero_mesa].Registro["DB919_Temporizadores_Registro_flujos".Temporizadores_mesa[#Numero_mesa].NUM_REGISTRO_ACTUAL].T_Giro, in11 := "DB920_Registro_Flujos".Mesa[#Numero_mesa].Registro["DB919_Temporizadores_Registro_flujos".Temporizadores_mesa[#Numero_mesa].NUM_REGISTRO_ACTUAL].T_Subir_Transfer, in12 := "DB920_Registro_Flujos".Mesa[#Numero_mesa].Registro["DB919_Temporizadores_Registro_flujos".Temporizadores_mesa[#Numero_mesa].NUM_REGISTRO_ACTUAL].T_Bajar_Transfer, out => "DB920_Registro_Flujos".Mesa[#Numero_mesa].Registro["DB919_Temporizadores_Registro_flujos".Temporizadores_mesa[#Numero_mesa].NUM_REGISTRO_ACTUAL].T_Total)
   END_RUNG
   // the same network as SCL:
   "DB920_Registro_Flujos".Mesa[#Numero_mesa].Registro["DB919_Temporizadores_Registro_flujos".Temporizadores_mesa[#Numero_mesa].NUM_REGISTRO_ACTUAL].T_Total := "DB920_Registro_Flujos".Mesa[#Numero_mesa].Registro["DB919_Temporizadores_Registro_flujos".Temporizadores_mesa[#Numero_mesa].NUM_REGISTRO_ACTUAL].T_Etapa_Carga_E1 + "DB920_Registro_Flujos".Mesa[#Numero_mesa].Registro["DB919_Temporizadores_Registro_flujos".Temporizadores_mesa[#Numero_mesa].NUM_REGISTRO_ACTUAL].T_Etapa_Carga_E2 + "DB920_Registro_Flujos".Mesa[#Numero_mesa].Registro["DB919_Temporizadores_Registro_flujos".Temporizadores_mesa[#Numero_mesa].NUM_REGISTRO_ACTUAL].T_Etapa_Carga_E3 + "DB920_Registro_Flujos".Mesa[#Numero_mesa].Registro["DB919_Temporizadores_Registro_flujos".Temporizadores_mesa[#Numero_mesa].NUM_REGISTRO_ACTUAL].T_Etapa_Carga_E4 + "DB920_Registro_Flujos".Mesa[#Numero_mesa].Registro["DB919_Temporizadores_Registro_flujos".Temporizadores_mesa[#Numero_mesa].NUM_REGISTRO_ACTUAL].T_Etapa_Cargada + "DB920_Registro_Flujos".Mesa[#Numero_mesa].Registro["DB919_Temporizadores_Registro_flujos".Temporizadores_mesa[#Numero_mesa].NUM_REGISTRO_ACTUAL].T_Etapa_Descarga_S1 + "DB920_Registro_Flujos".Mesa[#Numero_mesa].Registro["DB919_Temporizadores_Registro_flujos".Temporizadores_mesa[#Numero_mesa].NUM_REGISTRO_ACTUAL].T_Etapa_Descarga_S2 + "DB920_Registro_Flujos".Mesa[#Numero_mesa].Registro["DB919_Temporizadores_Registro_flujos".Temporizadores_mesa[#Numero_mesa].NUM_REGISTRO_ACTUAL].T_Etapa_Descarga_S3 + "DB920_Registro_Flujos".Mesa[#Numero_mesa].Registro["DB919_Temporizadores_Registro_flujos".Temporizadores_mesa[#Numero_mesa].NUM_REGISTRO_ACTUAL].T_Etapa_Descarga_S4 + "DB920_Registro_Flujos".Mesa[#Numero_mesa].Registro["DB919_Temporizadores_Registro_flujos".Temporizadores_mesa[#Numero_mesa].NUM_REGISTRO_ACTUAL].T_Giro + "DB920_Registro_Flujos".Mesa[#Numero_mesa].Registro["DB919_Temporizadores_Registro_flujos".Temporizadores_mesa[#Numero_mesa].NUM_REGISTRO_ACTUAL].T_Subir_Transfer + "DB920_Registro_Flujos".Mesa[#Numero_mesa].Registro["DB919_Temporizadores_Registro_flujos".Temporizadores_mesa[#Numero_mesa].NUM_REGISTRO_ACTUAL].T_Bajar_Transfer;
END_REGION
END_FUNCTION
